(* IEC 61131-3 sources: FB_Sequence/integration/service_v02, 7 files *)

(* ---- ST_SEQ_SVC_CONFIG.st ---- *)
TYPE ST_SEQ_SVC_CONFIG :
STRUCT
    xEnable : BOOL;
    uiServiceContractMajor : UINT;
    uiServiceContractMinor : UINT;
    udiMappingRevision : UDINT;
    uiExpectedMachineID : UINT;
    uiExpectedProducerSourceID : UINT;
    uiExpectedProcessID : UINT;
    udiProducerID : UDINT;
END_STRUCT
END_TYPE

(* ---- ST_SEQ_SVC_ENVELOPE.st ---- *)
TYPE ST_SEQ_SVC_ENVELOPE :
STRUCT
    udiMappingRevision : UDINT;
    xProjectionLossless : BOOL;
    // Authoritative, immutable source event. Never discard this sidecar.
    stSourceEvent : ST_SEQ_EVENT;
    // Searchable generic projection; intentionally not a full audit copy.
    stServiceEvent : ST_SVC_EventInput;
END_STRUCT
END_TYPE

(* ---- ST_SEQ_SVC_RECEIPT.st ---- *)
TYPE ST_SEQ_SVC_RECEIPT :
STRUCT
    // External consumer owns the FULL envelope, not just its Service projection.
    // This is not ST_SVC_AuditAck and is not generated by FB_Service v0.2.
    xValid : BOOL;
    xFullEnvelopeOwned : BOOL;
    udiMappingRevision : UDINT;
    uiMachineID : UINT;
    uiProducerSourceID : UINT;
    uiProcessID : UINT;
    udiSessionID : UDINT;
    udiEventID : UDINT;
END_STRUCT
END_TYPE

(* ---- ST_SEQ_SVC_SINK_RECEIPT.st ---- *)
TYPE ST_SEQ_SVC_SINK_RECEIPT :
STRUCT
    // Trusted sink owns the complete envelope AND binds it to this Service record.
    stSourceReceipt : ST_SEQ_SVC_RECEIPT;
    udiServiceBootID : UDINT;
    udiServiceRecordID : UDINT;
END_STRUCT
END_TYPE

(* ---- FB_SEQ_ServiceReceiptGate.st ---- *)
FUNCTION_BLOCK FB_SEQ_ServiceReceiptGate
VAR_INPUT
    xEnable : BOOL;
    xEnvelopeValid : BOOL;
    stEnvelope : ST_SEQ_SVC_ENVELOPE;
    stIngress : ST_SVC_EventReceipt;
    stSink : ST_SEQ_SVC_SINK_RECEIPT;
END_VAR
VAR_OUTPUT
    stReceipt : ST_SEQ_SVC_RECEIPT;
    xEligible : BOOL;
    xRejected : BOOL;
    xReadyForReceipt : BOOL; // Raw low observed for this eligible, unowned binding.
END_VAR
VAR
    stEmpty : ST_SEQ_SVC_RECEIPT;
    stOwnedReceipt : ST_SEQ_SVC_RECEIPT;
    stBoundIngress : ST_SVC_EventReceipt;
    udiBoundMapping : UDINT;
    xBound : BOOL;
    xArmed : BOOL;
    xOwned : BOOL;
    xSame : BOOL;
    xMatches : BOOL;
    xWasEligible : BOOL;
    xResume : BOOL;
END_VAR

// Optional receipt join; never sends commands, writes GVLs or removes either queue.
stReceipt := stEmpty;
xRejected := FALSE;
xEligible := xEnable AND xEnvelopeValid
    AND stEnvelope.stServiceEvent.xValid
    AND stEnvelope.stServiceEvent.stHeader.xValid
    AND (stEnvelope.udiMappingRevision <> UDINT#0)
    AND (stEnvelope.stSourceEvent.uiContractMajor = UINT#0)
    AND (stEnvelope.stSourceEvent.uiContractMinor = UINT#2)
    AND (stEnvelope.stSourceEvent.uiMachineID <> UINT#0)
    AND (stEnvelope.stSourceEvent.uiProducerSourceID <> UINT#0)
    AND (stEnvelope.stSourceEvent.uiProcessID <> UINT#0)
    AND (stEnvelope.stSourceEvent.udiSessionID <> UDINT#0)
    AND (stEnvelope.stSourceEvent.udiEventID <> UDINT#0)
    AND stIngress.xValid
    AND (stIngress.udiBootID <> UDINT#0)
    AND (stIngress.udiRecordID <> UDINT#0)
    AND (stIngress.uiMachineID = stEnvelope.stSourceEvent.uiMachineID)
    AND (stIngress.uiSourceID = stEnvelope.stSourceEvent.uiProducerSourceID)
    AND (stIngress.uiProcessID = stEnvelope.stSourceEvent.uiProcessID)
    AND (stIngress.udiSourceEpoch = stEnvelope.stSourceEvent.udiSessionID)
    AND (stIngress.udiSourceSeq = stEnvelope.stSourceEvent.udiEventID)
    AND (stIngress.uiSourceID = stEnvelope.stServiceEvent.stHeader.uiSourceID)
    AND (stIngress.uiProcessID = stEnvelope.stServiceEvent.stContext.uiProcessID)
    AND (stIngress.udiSourceEpoch = stEnvelope.stServiceEvent.stHeader.udiSourceEpoch)
    AND (stIngress.udiSourceSeq = stEnvelope.stServiceEvent.stHeader.udiSourceSeq);
xResume := xEligible AND NOT xWasEligible;
xWasEligible := xEligible;

IF NOT xEligible THEN
    // A masked output is NOT a low edge at the raw sink receipt input.
    xArmed := FALSE;
ELSE
    xSame := xBound
        AND (udiBoundMapping = stEnvelope.udiMappingRevision)
        AND (stBoundIngress.uiMachineID = stIngress.uiMachineID)
        AND (stBoundIngress.uiSourceID = stIngress.uiSourceID)
        AND (stBoundIngress.uiProcessID = stIngress.uiProcessID)
        AND (stBoundIngress.udiSourceEpoch = stIngress.udiSourceEpoch)
        AND (stBoundIngress.udiSourceSeq = stIngress.udiSourceSeq)
        AND (stBoundIngress.udiBootID = stIngress.udiBootID)
        AND (stBoundIngress.udiRecordID = stIngress.udiRecordID);
    IF NOT xSame THEN
        stBoundIngress := stIngress;
        udiBoundMapping := stEnvelope.udiMappingRevision;
        xBound := TRUE;
        xArmed := FALSE;
        xOwned := FALSE;
    END_IF;

    IF xOwned THEN
        // One low scan after regrant rearms a mapper that missed our prior receipt.
        // Ownership remains retained; do not invent a new sink transaction.
        IF NOT xResume THEN
            stReceipt := stOwnedReceipt;
        END_IF;
    ELSIF NOT stSink.stSourceReceipt.xValid THEN
        xArmed := TRUE;
    ELSE
        xMatches := stSink.stSourceReceipt.xFullEnvelopeOwned
            AND (stSink.udiServiceBootID = stBoundIngress.udiBootID)
            AND (stSink.udiServiceRecordID = stBoundIngress.udiRecordID)
            AND (stSink.stSourceReceipt.udiMappingRevision = udiBoundMapping)
            AND (stSink.stSourceReceipt.uiMachineID = stBoundIngress.uiMachineID)
            AND (stSink.stSourceReceipt.uiProducerSourceID = stBoundIngress.uiSourceID)
            AND (stSink.stSourceReceipt.uiProcessID = stBoundIngress.uiProcessID)
            AND (stSink.stSourceReceipt.udiSessionID = stBoundIngress.udiSourceEpoch)
            AND (stSink.stSourceReceipt.udiEventID = stBoundIngress.udiSourceSeq);
        IF xArmed AND xMatches THEN
            stOwnedReceipt := stSink.stSourceReceipt;
            xOwned := TRUE;
            stReceipt := stOwnedReceipt;
        ELSE
            xRejected := TRUE;
        END_IF;
        xArmed := FALSE;
    END_IF;
END_IF;
xReadyForReceipt := xEligible AND xArmed AND NOT xOwned;
END_FUNCTION_BLOCK

(* ---- FB_SEQ_ToServiceAdapter.st ---- *)
FUNCTION_BLOCK FB_SEQ_ToServiceAdapter
VAR_INPUT
    stCfg : ST_SEQ_SVC_CONFIG;
    xEventAvailable : BOOL;
    stEvent : ST_SEQ_EVENT;
    stReceipt : ST_SEQ_SVC_RECEIPT;
END_VAR
VAR_OUTPUT
    xEnvelopeValid : BOOL;
    stEnvelope : ST_SEQ_SVC_ENVELOPE;
    xConfigValid : BOOL;
    xSourceValid : BOOL;
    xPendingConflict : BOOL;
    xReceiptRejected : BOOL;
    xAck : BOOL;
    udiEventAckSessionID : UDINT;
    udiEventAckID : UDINT;
END_VAR
VAR
    stLatched : ST_SEQ_SVC_ENVELOPE;
    stEmpty : ST_SEQ_SVC_ENVELOPE;
    xPending : BOOL;
    xAckIssued : BOOL;
    xReceiptArmed : BOOL;
    xSameEvent : BOOL;
    xConfigMatches : BOOL;
    xReceiptMatches : BOOL;
    eDomain : E_SVC_Domain;
    eKind : E_SVC_EventKind;
    udiLatchedProducerID : UDINT;
END_VAR

// Pure software bridge. No Control/Sequence commands, output I/O or transport.
xEnvelopeValid := FALSE;
stEnvelope := stEmpty;
xAck := FALSE;
udiEventAckSessionID := UDINT#0;
udiEventAckID := UDINT#0;
xPendingConflict := FALSE;
xReceiptRejected := FALSE;

xConfigValid :=
    (stCfg.uiServiceContractMajor = UINT#2)
    AND (stCfg.uiServiceContractMinor = UINT#0)
    AND (stCfg.udiMappingRevision <> UDINT#0)
    AND (stCfg.uiExpectedMachineID <> UINT#0)
    AND (stCfg.uiExpectedProducerSourceID <> UINT#0)
    AND (stCfg.uiExpectedProcessID <> UINT#0)
    AND (stCfg.udiProducerID <> UDINT#0);

xSourceValid := xEventAvailable
    AND (stEvent.uiContractMajor = UINT#0)
    AND (stEvent.uiContractMinor = UINT#2)
    AND (stEvent.uiMachineID = stCfg.uiExpectedMachineID)
    AND (stEvent.uiProducerSourceID = stCfg.uiExpectedProducerSourceID)
    AND (stEvent.uiProcessID = stCfg.uiExpectedProcessID)
    AND (stEvent.udiSessionID <> UDINT#0)
    AND (stEvent.udiEventID <> UDINT#0);

eDomain := E_SVC_Domain.UNDEFINED;
eKind := E_SVC_EventKind.UNDEFINED;
CASE stEvent.eKind OF
    E_SEQ_EVENT_KIND.StateChanged:
        eDomain := E_SVC_Domain.PROCESS;
        eKind := E_SVC_EventKind.STATE_TRANSITION;
    E_SEQ_EVENT_KIND.StepChanged:
        eDomain := E_SVC_Domain.PROCESS;
        eKind := E_SVC_EventKind.CONTEXT_CHANGE;
    E_SEQ_EVENT_KIND.CommandResult:
        eDomain := E_SVC_Domain.PROCESS;
        eKind := E_SVC_EventKind.INTEGRATION;
    E_SEQ_EVENT_KIND.RecipeLoaded:
        eDomain := E_SVC_Domain.RECIPE;
        eKind := E_SVC_EventKind.CONTEXT_CHANGE;
    E_SEQ_EVENT_KIND.BatchStarted, E_SEQ_EVENT_KIND.BatchFinished:
        eDomain := E_SVC_Domain.BATCH;
        eKind := E_SVC_EventKind.BATCH_TRANSITION;
    E_SEQ_EVENT_KIND.StepStarted, E_SEQ_EVENT_KIND.StepFinished,
    E_SEQ_EVENT_KIND.PromptIssued, E_SEQ_EVENT_KIND.FaultRaised,
    E_SEQ_EVENT_KIND.FaultCleared:
        eDomain := E_SVC_Domain.PROCESS;
        eKind := E_SVC_EventKind.STATE_TRANSITION;
    E_SEQ_EVENT_KIND.PromptConfirmed, E_SEQ_EVENT_KIND.ResourceAcquired,
    E_SEQ_EVENT_KIND.ResourceReleased:
        eDomain := E_SVC_Domain.PROCESS;
        eKind := E_SVC_EventKind.INTEGRATION;
    E_SEQ_EVENT_KIND.RecipeRejected:
        eDomain := E_SVC_Domain.RECIPE;
        eKind := E_SVC_EventKind.INTEGRATION;
END_CASE;
xSourceValid := xSourceValid
    AND (eDomain <> E_SVC_Domain.UNDEFINED)
    AND (eKind <> E_SVC_EventKind.UNDEFINED);

xSameEvent := xPending
    AND (stLatched.stSourceEvent.uiMachineID = stEvent.uiMachineID)
    AND (stLatched.stSourceEvent.uiProducerSourceID = stEvent.uiProducerSourceID)
    AND (stLatched.stSourceEvent.uiProcessID = stEvent.uiProcessID)
    AND (stLatched.stSourceEvent.udiSessionID = stEvent.udiSessionID)
    AND (stLatched.stSourceEvent.udiEventID = stEvent.udiEventID);

IF NOT stCfg.xEnable OR NOT xConfigValid OR NOT xSourceValid THEN
    // Permission withdrawal suppresses output and ACK; retain pending privately.
    xReceiptArmed := FALSE;
ELSE
    IF (NOT xPending) OR (xAckIssued AND NOT xSameEvent) THEN
        stLatched := stEmpty;
        stLatched.udiMappingRevision := stCfg.udiMappingRevision;
        stLatched.xProjectionLossless := FALSE;
        stLatched.stSourceEvent := stEvent;
        // Unknown origin time keeps the full sidecar but blocks this projection.
        // Otherwise Service could replace it with ingestion time on collection.
        stLatched.stServiceEvent.xValid := stEvent.xOccurrenceTimeValid;
        stLatched.stServiceEvent.stHeader.xValid := stEvent.xOccurrenceTimeValid;
        stLatched.stServiceEvent.stHeader.uiSchemaMajor := stCfg.uiServiceContractMajor;
        stLatched.stServiceEvent.stHeader.uiSchemaMinor := stCfg.uiServiceContractMinor;
        stLatched.stServiceEvent.stHeader.uiSourceID := stEvent.uiProducerSourceID;
        stLatched.stServiceEvent.stHeader.eProducerKind := E_SVC_ActorKind.SEQUENCE_SOURCE;
        stLatched.stServiceEvent.stHeader.udiProducerID := stCfg.udiProducerID;
        stLatched.stServiceEvent.stHeader.udiSourceEpoch := stEvent.udiSessionID;
        stLatched.stServiceEvent.stHeader.udiSourceSeq := stEvent.udiEventID;
        stLatched.stServiceEvent.stHeader.udiTickMs := stEvent.udiOccurrenceTickMs;
        stLatched.stServiceEvent.stHeader.eQuality := E_SVC_DataQuality.GOOD;
        IF stEvent.xSyntheticTime OR NOT stEvent.xOccurrenceTimeValid THEN
            stLatched.stServiceEvent.stHeader.eQuality := E_SVC_DataQuality.UNCERTAIN;
        END_IF;
        // Valid here means the origin supplied its monotonic time, NOT valid UTC.
        stLatched.stServiceEvent.stTime.xValid := stEvent.xOccurrenceTimeValid;
        stLatched.stServiceEvent.stTime.udiTickMs := stEvent.udiOccurrenceTickMs;
        stLatched.stServiceEvent.stTime.eQuality := E_SVC_TimeQuality.UNSYNCHRONIZED;
        // UTC, clock source and authenticated actor remain zero/unknown.
        stLatched.stServiceEvent.stContext.udiBatchID := stEvent.udiBatchID;
        stLatched.stServiceEvent.stContext.udiRecipeID := stEvent.udiRecipeID;
        stLatched.stServiceEvent.stContext.udiRecipeRevision := stEvent.udiRecipeRevision;
        stLatched.stServiceEvent.stContext.uiProcessID := stEvent.uiProcessID;
        stLatched.stServiceEvent.stContext.uiStepID := stEvent.uiStepID;
        stLatched.stServiceEvent.eDomain := eDomain;
        stLatched.stServiceEvent.eKind := eKind;
        stLatched.stServiceEvent.uiObjectID := stEvent.uiProcessID;
        stLatched.stServiceEvent.uiEventCode := TO_UINT(stEvent.eKind);
        stLatched.stServiceEvent.uiReasonID := TO_UINT(stEvent.eReason);
        stLatched.stServiceEvent.eActorKind := E_SVC_ActorKind.UNKNOWN;
        stLatched.stServiceEvent.udiCorrelationID := stEvent.udiRequestID;
        stLatched.stServiceEvent.dwOldState := TO_DWORD(stEvent.eStateBefore);
        stLatched.stServiceEvent.dwNewState := TO_DWORD(stEvent.eState);
        stLatched.stServiceEvent.diOldValue := UINT_TO_DINT(stEvent.uiStepIDBefore);
        stLatched.stServiceEvent.diNewValue := UINT_TO_DINT(stEvent.uiStepID);
        udiLatchedProducerID := stCfg.udiProducerID;
        xPending := TRUE;
        xAckIssued := FALSE;
        xReceiptArmed := FALSE;
        xSameEvent := TRUE;
    END_IF;

    xConfigMatches :=
        (stLatched.udiMappingRevision = stCfg.udiMappingRevision)
        AND (stLatched.stServiceEvent.stHeader.uiSchemaMajor = stCfg.uiServiceContractMajor)
        AND (stLatched.stServiceEvent.stHeader.uiSchemaMinor = stCfg.uiServiceContractMinor)
        AND (udiLatchedProducerID = stCfg.udiProducerID);
    xPendingConflict := NOT xSameEvent OR NOT xConfigMatches;

    IF xPendingConflict THEN
        // Never overwrite an unowned event with another source head/config.
        xReceiptArmed := FALSE;
    ELSIF xAckIssued THEN
        // Hold/retry the exact already-owned head until the source advances.
        // This survives an ACK missed at a task/publication boundary.
        xAck := TRUE;
        udiEventAckSessionID := stLatched.stSourceEvent.udiSessionID;
        udiEventAckID := stLatched.stSourceEvent.udiEventID;
    ELSIF NOT xAckIssued THEN
        stEnvelope := stLatched;
        xEnvelopeValid := TRUE;
        IF NOT stReceipt.xValid THEN
            xReceiptArmed := TRUE;
        ELSE
            xReceiptMatches := stReceipt.xFullEnvelopeOwned
                AND (stReceipt.udiMappingRevision = stLatched.udiMappingRevision)
                AND (stReceipt.uiMachineID = stLatched.stSourceEvent.uiMachineID)
                AND (stReceipt.uiProducerSourceID = stLatched.stSourceEvent.uiProducerSourceID)
                AND (stReceipt.uiProcessID = stLatched.stSourceEvent.uiProcessID)
                AND (stReceipt.udiSessionID = stLatched.stSourceEvent.udiSessionID)
                AND (stReceipt.udiEventID = stLatched.stSourceEvent.udiEventID);
            IF xReceiptArmed AND xReceiptMatches THEN
                xAck := TRUE;
                udiEventAckSessionID := stLatched.stSourceEvent.udiSessionID;
                udiEventAckID := stLatched.stSourceEvent.udiEventID;
                xAckIssued := TRUE;
            ELSE
                xReceiptRejected := TRUE;
            END_IF;
            xReceiptArmed := FALSE;
        END_IF;
    END_IF;
END_IF;
END_FUNCTION_BLOCK

(* ---- PRG_SEQ_ServiceBench.st ---- *)
// OFFLINE SIMULATOR ONLY. Independent instances; no GVL, I/O or network writer.
// Select this program alone in one cyclic simulation task. Native execution is pending.
PROGRAM PRG_SEQ_ServiceBench
VAR
    xEnableBench : BOOL := FALSE;
    xAllowRequests : BOOL := FALSE;
    xAllowExecution : BOOL := FALSE;
    xAllowPublication : BOOL := FALSE;
    xQualified : BOOL := FALSE;
    xStepComplete : BOOL := FALSE;
    xFinishActions : BOOL := FALSE;
    xMockFaulted : BOOL := FALSE;
    xMockRejectRequest : BOOL := FALSE;
    udiAuthorityID : UDINT := 17;
    stSequenceCfg : ST_SEQ_CONFIG := (uiProcessID := 7, udiSessionID := 1001,
        udiMaxFeedbackAgeMs := 250, udiTransitionTimeoutMs := 5000,
        udiMaxCycleMs := 100, uiMachineID := 1, uiProducerSourceID := 301);
    stMapCfg : ST_SEQ_SVC_CONFIG := (uiServiceContractMajor := 2,
        uiServiceContractMinor := 0, udiMappingRevision := 1,
        uiExpectedMachineID := 1, uiExpectedProducerSourceID := 301,
        uiExpectedProcessID := 7, udiProducerID := 301);
    stServiceCfg : ST_SVC_Config;
    stTraceTime : ST_SEQ_TRACE_TIME;
    stServiceTime : ST_SVC_TimeContext;
    stCommand : ST_SEQ_COMMAND_REQUEST;
    stRecipe : ST_SEQ_RECIPE;
    // The sole external writer may copy the ACTUAL sink receipt after file COMMIT.
    // First observe this raw receipt invalid while xCaptureReady; never synthesize ownership.
    stSinkReturned : ST_SEQ_SVC_SINK_RECEIPT;
    // Separate audit channel: no value is derived from source/sink receipt.
    stAuditAck : ST_SVC_AuditAck;
    stRuntimeUnknown : ST_SVC_RuntimeInput;
    stOperationsUnknown : ST_SVC_OperationsInput;
    aAlarmUnknown : ARRAY[1..16] OF ST_SVC_AlarmCondition;
    aEvents : ARRAY[1..8] OF ST_SVC_EventInput;
    stNoEvent : ST_SVC_EventInput;
    stCaptureEnvelope : ST_SEQ_SVC_ENVELOPE;
    stCaptureIngress : ST_SVC_EventReceipt;
    stEmptyEnvelope : ST_SEQ_SVC_ENVELOPE;
    stEmptyIngress : ST_SVC_EventReceipt;
    xCaptureReady : BOOL;
    xPublicationAllowed : BOOL;
    udiSourceAckSession : UDINT;
    udiSourceAckEvent : UDINT;
    fbControlMock : FB_SEQ_ControlMock;
    fbSequence : FB_Sequence;
    fbMapper : FB_SEQ_ToServiceAdapter;
    fbService : FB_Service;
    fbReceiptGate : FB_SEQ_ServiceReceiptGate;
    xInitialized : BOOL;
END_VAR

IF NOT xInitialized THEN
    stServiceCfg.uiContractMajor := UINT#2;
    stServiceCfg.uiContractMinor := UINT#0;
    stServiceCfg.udiConfigRevision := UDINT#1;
    stServiceCfg.udiBootID := UDINT#2002;
    stServiceCfg.uiServiceSourceID := UINT#900;
    stServiceCfg.stAsset.uiMachineID := UINT#1;
    stServiceCfg.stAsset.uiWorkUnitID := UINT#1;
    stServiceCfg.udiRuntimeFreshnessMs := UDINT#500;
    stServiceCfg.udiOperationsFreshnessMs := UDINT#500;
    stServiceCfg.udiAlarmFreshnessMs := UDINT#500;
    // No OEE or equipment facts are invented for this event-only composition.
    stServiceCfg.stOEEPolicy.xEnabled := FALSE;
    stRecipe.udiRecipeID := UDINT#1;
    stRecipe.udiRevision := UDINT#1;
    stRecipe.uiStepCount := UINT#1;
    stRecipe.astSteps[1].uiStepID := UINT#10;
    stRecipe.astSteps[1].uiPhaseID := UINT#10;
    stRecipe.astSteps[1].uiProfileID := UINT#100;
    stRecipe.astSteps[1].eKind := E_SEQ_STEP_KIND.WaitQualified;
    stRecipe.astSteps[1].udiQualifiedMs := UDINT#250;
    stRecipe.astSteps[1].udiTimeoutMs := UDINT#10000;
    xInitialized := TRUE;
END_IF;

stTraceTime.udiTickMs := F_SEQ_AddMs(stTraceTime.udiTickMs, UDINT#20);
stTraceTime.xValid := stTraceTime.udiTickMs < UDINT#4294967295;
stTraceTime.xSynthetic := TRUE;
stServiceTime.xValid := stTraceTime.xValid;
stServiceTime.udiTickMs := stTraceTime.udiTickMs;
stServiceTime.eQuality := E_SVC_TimeQuality.UNSYNCHRONIZED;

// Previous scan's request enters the Control test double, which owns permissions.
fbControlMock(xEnable := xEnableBench, stRequest := fbSequence.stControlRequest,
    stConfig := stSequenceCfg, xAllowRequests := xAllowRequests,
    xAllowExecution := xAllowExecution, xAllowPublication := xAllowPublication,
    xQualified := xQualified, xStepComplete := xStepComplete,
    xFaulted := xMockFaulted, xRejectRequest := xMockRejectRequest,
    xFinishActions := xFinishActions, udiAuthorityID := udiAuthorityID);
xPublicationAllowed := xEnableBench AND fbControlMock.stAuthority.xValid
    AND fbControlMock.stAuthority.xAllowPublication
    AND (fbControlMock.stAuthority.udiSessionID = stSequenceCfg.udiSessionID)
    AND (fbControlMock.stAuthority.uiProcessID = stSequenceCfg.uiProcessID)
    AND (fbControlMock.stAuthority.udiAuthorityID <> UDINT#0)
    AND (fbControlMock.stAuthority.udiAgeMs <= stSequenceCfg.udiMaxFeedbackAgeMs);

// Only the previous mapper output is a source ACK, and only under current publication permission.
udiSourceAckSession := UDINT#0;
udiSourceAckEvent := UDINT#0;
IF xPublicationAllowed AND fbMapper.xAck THEN
    udiSourceAckSession := fbMapper.udiEventAckSessionID;
    udiSourceAckEvent := fbMapper.udiEventAckID;
END_IF;
fbSequence(xEnable := xEnableBench, stConfig := stSequenceCfg,
    udiDeltaMs := UDINT#20, stTraceTime := stTraceTime,
    stCommand := stCommand, stRecipeCandidate := stRecipe,
    stAuthority := fbControlMock.stAuthority, stControlResult := fbControlMock.stResult,
    stControlRuntime := fbControlMock.stRuntime,
    udiEventAckSessionID := udiSourceAckSession, udiEventAckID := udiSourceAckEvent);

// One mapper call per scan. Its receipt input is the gate's previous scan output.
stMapCfg.xEnable := xPublicationAllowed;
fbMapper(stCfg := stMapCfg, xEventAvailable := fbSequence.xEventAvailable,
    stEvent := fbSequence.stEvent, stReceipt := fbReceiptGate.stReceipt);
aEvents[1] := stNoEvent;
IF fbMapper.xEnvelopeValid THEN
    // Level held, immutable, fixed producer slot 1 until ownership is confirmed.
    aEvents[1] := fbMapper.stEnvelope.stServiceEvent;
END_IF;
stServiceCfg.xEnabled := xEnableBench;
fbService(stCfg := stServiceCfg, stTime := stServiceTime,
    stRuntime := stRuntimeUnknown, stOperations := stOperationsUnknown,
    aAlarmConditions := aAlarmUnknown, aEvents := aEvents,
    stAuditAck := stAuditAck, xResetOEEWindow := FALSE, udiNextOEEWindowID := UDINT#0);
fbReceiptGate(xEnable := xPublicationAllowed,
    xEnvelopeValid := fbMapper.xEnvelopeValid, stEnvelope := fbMapper.stEnvelope,
    stIngress := fbService.aEventReceipts[1], stSink := stSinkReturned);

// Same-task export view: capture these two complete structures together.
// An IDE/platform exporter must still be validated; this POU does not serialize files.
xCaptureReady := fbReceiptGate.xEligible;
stCaptureEnvelope := stEmptyEnvelope;
stCaptureIngress := stEmptyIngress;
IF xCaptureReady THEN
    stCaptureEnvelope := fbMapper.stEnvelope;
    stCaptureIngress := fbService.aEventReceipts[1];
END_IF;
END_PROGRAM
